FUNCTION_BLOCK FB_FanControl_Test EXTENDS FB_TestSuite
VAR
END_VAR

FanSpeedMax();
FanSpeedZero();

METHOD FanSpeedMax
VAR
	fbFanControl : FB_FanControl;		//Function Block call
	FanControlRes : INT;				//Actual value of FanControl
	ExpectedValue : INT := 32767;		//Expected value for FanControl
END_VAR
TEST('FanSpeedMax');
 
fbFanControl.fSpeed := 100;
fbFanControl();
FanControlRes := fbFanControl.fSpeedSetRaw;
 
AssertEquals(Expected := ExpectedValue,
             Actual := FanControlRes,
             Message := 'The calculation is not correct');
 
TEST_FINISHED();
END_METHOD

METHOD FanSpeedZero
VAR
	fbFanControl : FB_FanControl;		//Function Block call
	FanControlRes : INT;				//Actual value of FanControl
	ExpectedValue : INT := 0;			//Expected value for FanControl

END_VAR
TEST('FanSpeedZero');
 
fbFanControl.fSpeed := 0;
fbFanControl();
FanControlRes := fbFanControl.fSpeedSetRaw;
 
AssertEquals(Expected := ExpectedValue,
             Actual := FanControlRes,
             Message := 'The calculation is not correct');
 
TEST_FINISHED();
END_METHOD

END_FUNCTION_BLOCK

(* stored: Version 1.1.0.1, ProductVersion 3.1.4024.6
   POU FB_FanControl_Test: Id {d336d90e-9b76-4ab1-86b2-59be1e37978b}, SpecialFunc None
   Method FanSpeedMax: Id {cba8bbbb-a15f-4112-9849-e0b4cc86d529}
   Method FanSpeedZero: Id {737b7d60-6078-45b6-9461-42c67f132871} *)
